# EPICS substitutions: hugo/source/db/Beckhoff_3XXX/ecmcEL3602.substitutions
file "ecmc_analogInput-chX.template"
{
  pattern {CH_ID, ESLO,           EOFF, EGU, PREC}
          {01,    4.656612875E-9, 0,    "V", 3   }
          {02,    4.656612875E-9, 0,    "V", 3   }
}

file "ecmc_status-chX.template"
{
  pattern {CH_ID, KEY }
          {01,    "AI"}
          {02,    "AI"}
}
